PROGRAM P_Light_Test_ST
VAR
	fbLight				:	FB_Light;
	bOn					:	BOOL;
	bOff				:	BOOL;
	bControlLevel		:	BOOL;	
END_VAR

fbLight();

IF (bOn) THEN
	fbLight.M_On();
	bOn := FALSE;
END_IF
IF (bOff) THEN
	fbLight.M_Off();
	bOff := FALSE;
END_IF

bControlLevel := fbLight.bControlLevel;

END_PROGRAM

(* stored: Version 1.1.0.1, ProductVersion 3.1.4024.12
   POU P_Light_Test_ST: Id {2dc43587-1fdb-406e-a556-9521154ef615}, SpecialFunc None *)
